// TIA Portal V19 export
FUNCTION "OUTPUT MAPPING" : Void   // FC2, LAD
{ S7_Optimized_Access := 'TRUE' }
// stored: SetENOAutomatically false
BEGIN

REGION Network 1: "HOOTER RESET"
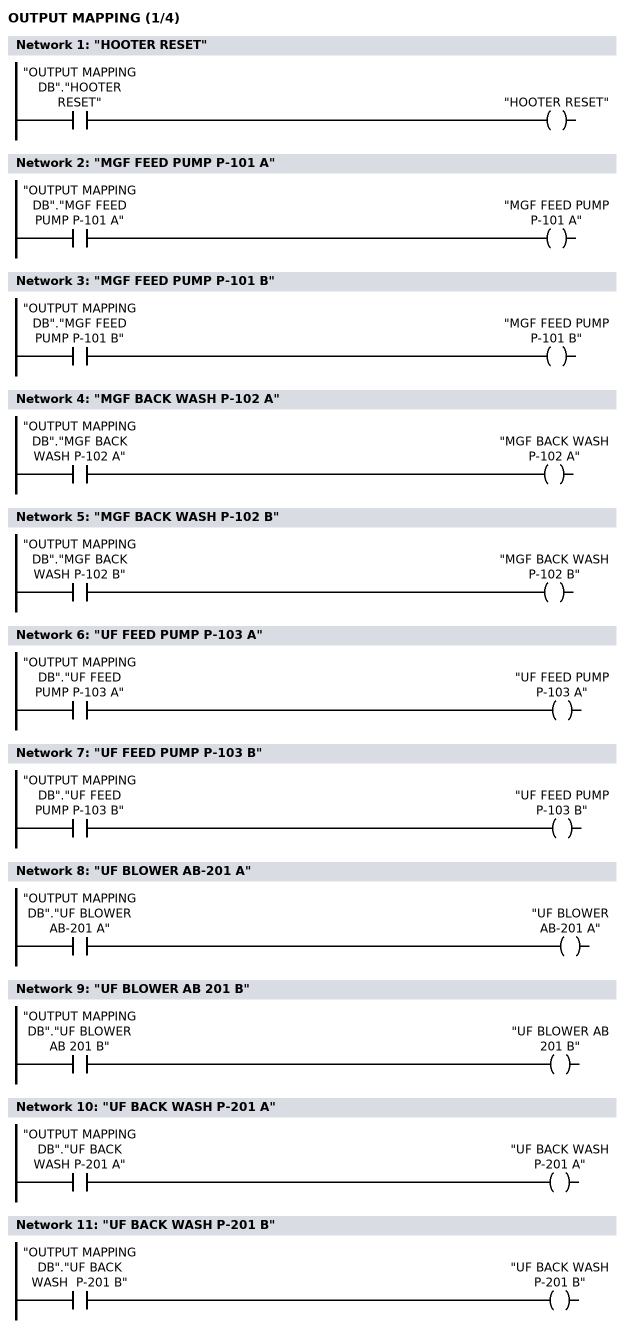
   RUNG wire#powerrail
      Contact( "OUTPUT MAPPING DB"."HOOTER RESET" )
      Coil( "HOOTER RESET" )
   END_RUNG
   // the same network as SCL:
   "HOOTER RESET" := "OUTPUT MAPPING DB"."HOOTER RESET";
END_REGION

REGION Network 2: "MGF FEED PUMP P-101 A"
   RUNG wire#powerrail
      Contact( "OUTPUT MAPPING DB"."MGF FEED PUMP P-101 A" )
      Coil( "MGF FEED PUMP P-101 A" )
   END_RUNG
   // the same network as SCL:
   "MGF FEED PUMP P-101 A" := "OUTPUT MAPPING DB"."MGF FEED PUMP P-101 A";
END_REGION

REGION Network 3: "MGF FEED PUMP P-101 B"
   RUNG wire#powerrail
      Contact( "OUTPUT MAPPING DB"."MGF FEED PUMP P-101 B" )
      Coil( "MGF FEED PUMP P-101 B" )
   END_RUNG
   // the same network as SCL:
   "MGF FEED PUMP P-101 B" := "OUTPUT MAPPING DB"."MGF FEED PUMP P-101 B";
END_REGION

REGION Network 4: "MGF BACK WASH P-102 A"
   RUNG wire#powerrail
      Contact( "OUTPUT MAPPING DB"."MGF BACK WASH P-102 A" )
      Coil( "MGF BACK WASH P-102 A" )
   END_RUNG
   // the same network as SCL:
   "MGF BACK WASH P-102 A" := "OUTPUT MAPPING DB"."MGF BACK WASH P-102 A";
END_REGION

REGION Network 5: "MGF BACK WASH P-102 B"
   RUNG wire#powerrail
      Contact( "OUTPUT MAPPING DB"."MGF BACK WASH P-102 B" )
      Coil( "MGF BACK WASH P-102 B" )
   END_RUNG
   // the same network as SCL:
   "MGF BACK WASH P-102 B" := "OUTPUT MAPPING DB"."MGF BACK WASH P-102 B";
END_REGION

REGION Network 6: "UF FEED PUMP P-103 A"
   RUNG wire#powerrail
      Contact( "OUTPUT MAPPING DB"."UF FEED PUMP P-103 A" )
      Coil( "UF FEED PUMP P-103 A" )
   END_RUNG
   // the same network as SCL:
   "UF FEED PUMP P-103 A" := "OUTPUT MAPPING DB"."UF FEED PUMP P-103 A";
END_REGION

REGION Network 7: "UF FEED PUMP P-103 B"
   RUNG wire#powerrail
      Contact( "OUTPUT MAPPING DB"."UF FEED PUMP P-103 B" )
      Coil( "UF FEED PUMP P-103 B" )
   END_RUNG
   // the same network as SCL:
   "UF FEED PUMP P-103 B" := "OUTPUT MAPPING DB"."UF FEED PUMP P-103 B";
END_REGION

REGION Network 8: "UF BLOWER AB-201 A"
   RUNG wire#powerrail
      Contact( "OUTPUT MAPPING DB"."UF BLOWER AB-201 A" )
      Coil( "UF BLOWER AB-201 A" )
   END_RUNG
   // the same network as SCL:
   "UF BLOWER AB-201 A" := "OUTPUT MAPPING DB"."UF BLOWER AB-201 A";
END_REGION

REGION Network 9: "UF BLOWER AB 201 B"
   RUNG wire#powerrail
      Contact( "OUTPUT MAPPING DB"."UF BLOWER AB 201 B" )
      Coil( "UF BLOWER AB 201 B" )
   END_RUNG
   // the same network as SCL:
   "UF BLOWER AB 201 B" := "OUTPUT MAPPING DB"."UF BLOWER AB 201 B";
END_REGION

REGION Network 10: "UF BACK WASH P-201 A"
   RUNG wire#powerrail
      Contact( "OUTPUT MAPPING DB"."UF BACK WASH P-201 A" )
      Coil( "UF BACK WASH P-201 A" )
   END_RUNG
   // the same network as SCL:
   "UF BACK WASH P-201 A" := "OUTPUT MAPPING DB"."UF BACK WASH P-201 A";
END_REGION

REGION Network 11: "UF BACK WASH P-201 B"
   RUNG wire#powerrail
      Contact( "OUTPUT MAPPING DB"."UF BACK WASH  P-201 B" )
      Coil( "UF BACK WASH  P-201 B" )
   END_RUNG
   // the same network as SCL:
   "UF BACK WASH  P-201 B" := "OUTPUT MAPPING DB"."UF BACK WASH  P-201 B";
END_REGION

REGION Network 12: "DM FEED PUMP P-502 A"
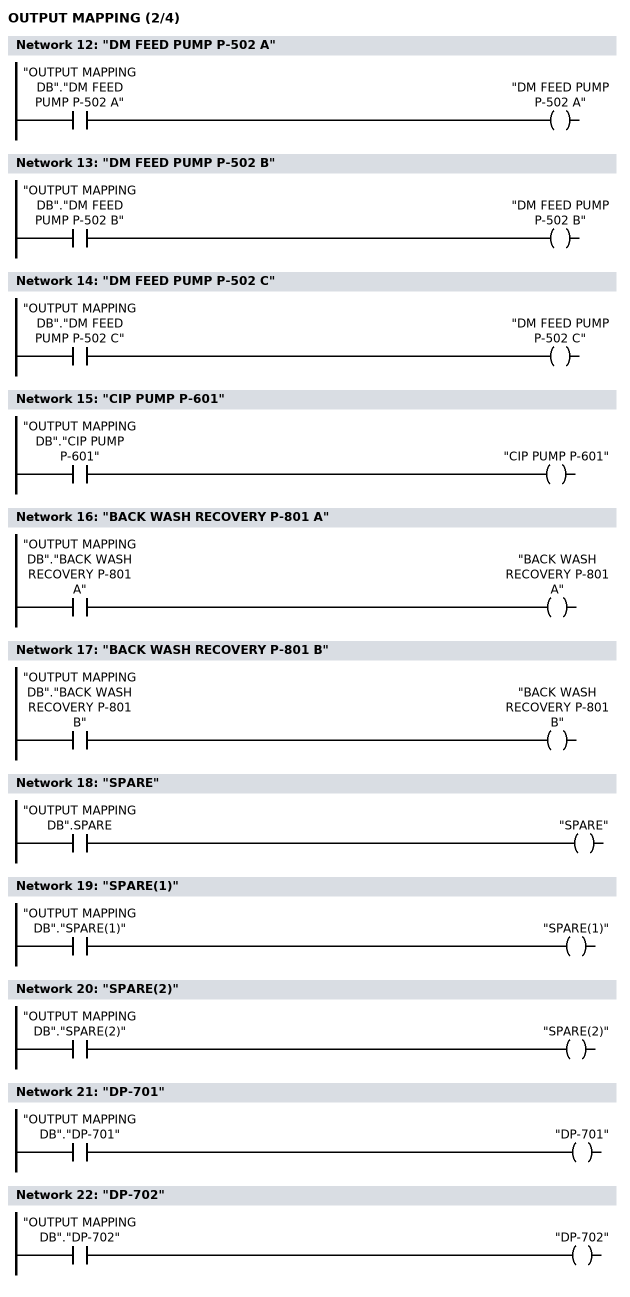
   RUNG wire#powerrail
      Contact( "OUTPUT MAPPING DB"."DM FEED PUMP P-502 A" )
      Coil( "DM FEED PUMP P-502 A" )
   END_RUNG
   // the same network as SCL:
   "DM FEED PUMP P-502 A" := "OUTPUT MAPPING DB"."DM FEED PUMP P-502 A";
END_REGION

REGION Network 13: "DM FEED PUMP P-502 B"
   RUNG wire#powerrail
      Contact( "OUTPUT MAPPING DB"."DM FEED PUMP P-502 B" )
      Coil( "DM FEED PUMP P-502 B" )
   END_RUNG
   // the same network as SCL:
   "DM FEED PUMP P-502 B" := "OUTPUT MAPPING DB"."DM FEED PUMP P-502 B";
END_REGION

REGION Network 14: "DM FEED PUMP P-502 C"
   RUNG wire#powerrail
      Contact( "OUTPUT MAPPING DB"."DM FEED PUMP P-502 C" )
      Coil( "DM FEED PUMP P-502 C" )
   END_RUNG
   // the same network as SCL:
   "DM FEED PUMP P-502 C" := "OUTPUT MAPPING DB"."DM FEED PUMP P-502 C";
END_REGION

REGION Network 15: "CIP PUMP P-601"
   RUNG wire#powerrail
      Contact( "OUTPUT MAPPING DB"."CIP PUMP P-601" )
      Coil( "CIP PUMP P-601" )
   END_RUNG
   // the same network as SCL:
   "CIP PUMP P-601" := "OUTPUT MAPPING DB"."CIP PUMP P-601";
END_REGION

REGION Network 16: "BACK WASH RECOVERY P-801 A"
   RUNG wire#powerrail
      Contact( "OUTPUT MAPPING DB"."BACK WASH RECOVERY P-801 A" )
      Coil( "BACK WASH RECOVERY P-801 A" )
   END_RUNG
   // the same network as SCL:
   "BACK WASH RECOVERY P-801 A" := "OUTPUT MAPPING DB"."BACK WASH RECOVERY P-801 A";
END_REGION

REGION Network 17: "BACK WASH RECOVERY P-801 B"
   RUNG wire#powerrail
      Contact( "OUTPUT MAPPING DB"."BACK WASH RECOVERY P-801 B" )
      Coil( "BACK WASH RECOVERY P-801 B" )
   END_RUNG
   // the same network as SCL:
   "BACK WASH RECOVERY P-801 B" := "OUTPUT MAPPING DB"."BACK WASH RECOVERY P-801 B";
END_REGION

REGION Network 18: "SPARE"
   RUNG wire#powerrail
      Contact( "OUTPUT MAPPING DB".SPARE )
      Coil( "SPARE" )
   END_RUNG
   // the same network as SCL:
   "SPARE" := "OUTPUT MAPPING DB".SPARE;
END_REGION

REGION Network 19: "SPARE(1)"
   RUNG wire#powerrail
      Contact( "OUTPUT MAPPING DB"."SPARE(1)" )
      Coil( "SPARE(1)" )
   END_RUNG
   // the same network as SCL:
   "SPARE(1)" := "OUTPUT MAPPING DB"."SPARE(1)";
END_REGION

REGION Network 20: "SPARE(2)"
   RUNG wire#powerrail
      Contact( "OUTPUT MAPPING DB"."SPARE(2)" )
      Coil( "SPARE(2)" )
   END_RUNG
   // the same network as SCL:
   "SPARE(2)" := "OUTPUT MAPPING DB"."SPARE(2)";
END_REGION

REGION Network 21: "DP-701"
   RUNG wire#powerrail
      Contact( "OUTPUT MAPPING DB"."DP-701" )
      Coil( "DP-701" )
   END_RUNG
   // the same network as SCL:
   "DP-701" := "OUTPUT MAPPING DB"."DP-701";
END_REGION

REGION Network 22: "DP-702"
   RUNG wire#powerrail
      Contact( "OUTPUT MAPPING DB"."DP-702" )
      Coil( "DP-702" )
   END_RUNG
   // the same network as SCL:
   "DP-702" := "OUTPUT MAPPING DB"."DP-702";
END_REGION

REGION Network 23: "NaOCL DOSING D-706 A"
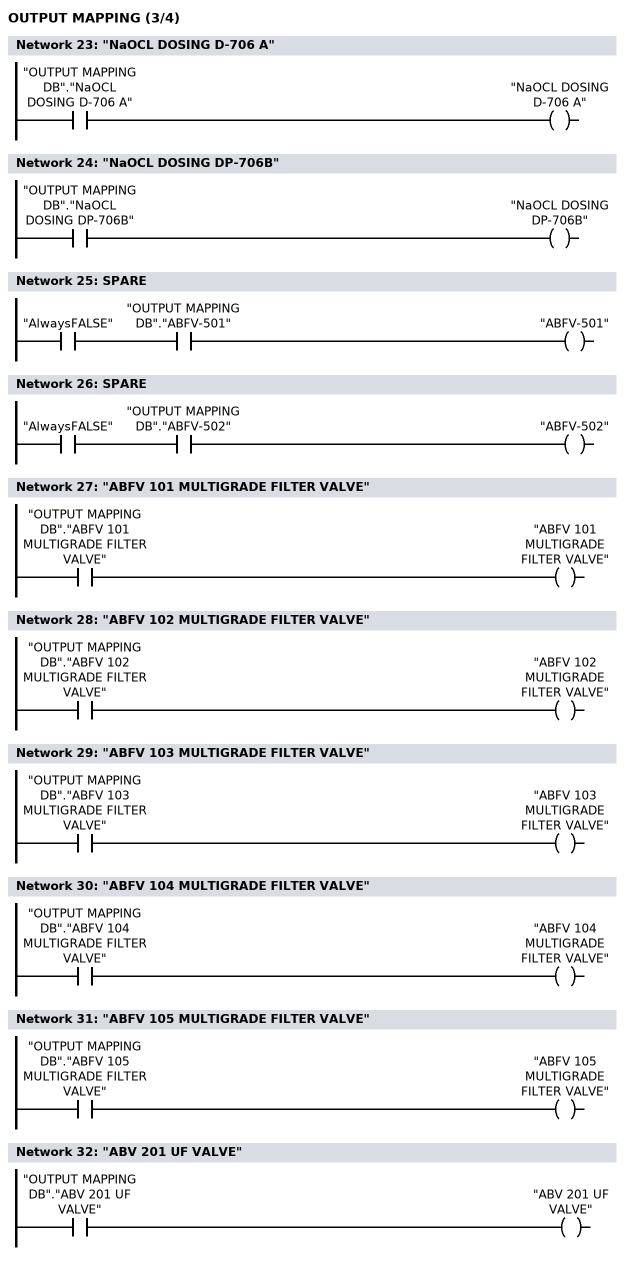
   RUNG wire#powerrail
      Contact( "OUTPUT MAPPING DB"."NaOCL DOSING D-706 A" )
      Coil( "NaOCL DOSING D-706 A" )
   END_RUNG
   // the same network as SCL:
   "NaOCL DOSING D-706 A" := "OUTPUT MAPPING DB"."NaOCL DOSING D-706 A";
END_REGION

REGION Network 24: "NaOCL DOSING DP-706B"
   RUNG wire#powerrail
      Contact( "OUTPUT MAPPING DB"."NaOCL DOSING DP-706B" )
      Coil( "NaOCL DOSING DP-706B" )
   END_RUNG
   // the same network as SCL:
   "NaOCL DOSING DP-706B" := "OUTPUT MAPPING DB"."NaOCL DOSING DP-706B";
END_REGION

REGION Network 25: SPARE
   RUNG wire#powerrail
      Contact( "AlwaysFALSE" )
      Contact( "OUTPUT MAPPING DB"."ABFV-501" )
      Coil( "ABFV-501" )
   END_RUNG
   // the same network as SCL:
   "ABFV-501" := "AlwaysFALSE" AND "OUTPUT MAPPING DB"."ABFV-501";
END_REGION

REGION Network 26: SPARE
   RUNG wire#powerrail
      Contact( "AlwaysFALSE" )
      Contact( "OUTPUT MAPPING DB"."ABFV-502" )
      Coil( "ABFV-502" )
   END_RUNG
   // the same network as SCL:
   "ABFV-502" := "AlwaysFALSE" AND "OUTPUT MAPPING DB"."ABFV-502";
END_REGION

REGION Network 27: "ABFV 101 MULTIGRADE FILTER VALVE"
   RUNG wire#powerrail
      Contact( "OUTPUT MAPPING DB"."ABFV 101 MULTIGRADE FILTER VALVE" )
      Coil( "ABFV 101 MULTIGRADE FILTER VALVE" )
   END_RUNG
   // the same network as SCL:
   "ABFV 101 MULTIGRADE FILTER VALVE" := "OUTPUT MAPPING DB"."ABFV 101 MULTIGRADE FILTER VALVE";
END_REGION

REGION Network 28: "ABFV 102 MULTIGRADE FILTER VALVE"
   RUNG wire#powerrail
      Contact( "OUTPUT MAPPING DB"."ABFV 102 MULTIGRADE FILTER VALVE" )
      Coil( "ABFV 102 MULTIGRADE FILTER VALVE" )
   END_RUNG
   // the same network as SCL:
   "ABFV 102 MULTIGRADE FILTER VALVE" := "OUTPUT MAPPING DB"."ABFV 102 MULTIGRADE FILTER VALVE";
END_REGION

REGION Network 29: "ABFV 103 MULTIGRADE FILTER VALVE"
   RUNG wire#powerrail
      Contact( "OUTPUT MAPPING DB"."ABFV 103 MULTIGRADE FILTER VALVE" )
      Coil( "ABFV 103 MULTIGRADE FILTER VALVE" )
   END_RUNG
   // the same network as SCL:
   "ABFV 103 MULTIGRADE FILTER VALVE" := "OUTPUT MAPPING DB"."ABFV 103 MULTIGRADE FILTER VALVE";
END_REGION

REGION Network 30: "ABFV 104 MULTIGRADE FILTER VALVE"
   RUNG wire#powerrail
      Contact( "OUTPUT MAPPING DB"."ABFV 104 MULTIGRADE FILTER VALVE" )
      Coil( "ABFV 104 MULTIGRADE FILTER VALVE" )
   END_RUNG
   // the same network as SCL:
   "ABFV 104 MULTIGRADE FILTER VALVE" := "OUTPUT MAPPING DB"."ABFV 104 MULTIGRADE FILTER VALVE";
END_REGION

REGION Network 31: "ABFV 105 MULTIGRADE FILTER VALVE"
   RUNG wire#powerrail
      Contact( "OUTPUT MAPPING DB"."ABFV 105 MULTIGRADE FILTER VALVE" )
      Coil( "ABFV 105 MULTIGRADE FILTER VALVE" )
   END_RUNG
   // the same network as SCL:
   "ABFV 105 MULTIGRADE FILTER VALVE" := "OUTPUT MAPPING DB"."ABFV 105 MULTIGRADE FILTER VALVE";
END_REGION

REGION Network 32: "ABV 201 UF VALVE"
   RUNG wire#powerrail
      Contact( "OUTPUT MAPPING DB"."ABV 201 UF VALVE" )
      Coil( "ABV 201 UF VALVE" )
   END_RUNG
   // the same network as SCL:
   "ABV 201 UF VALVE" := "OUTPUT MAPPING DB"."ABV 201 UF VALVE";
END_REGION

REGION Network 33: "ABFV 201 UF VALVE"
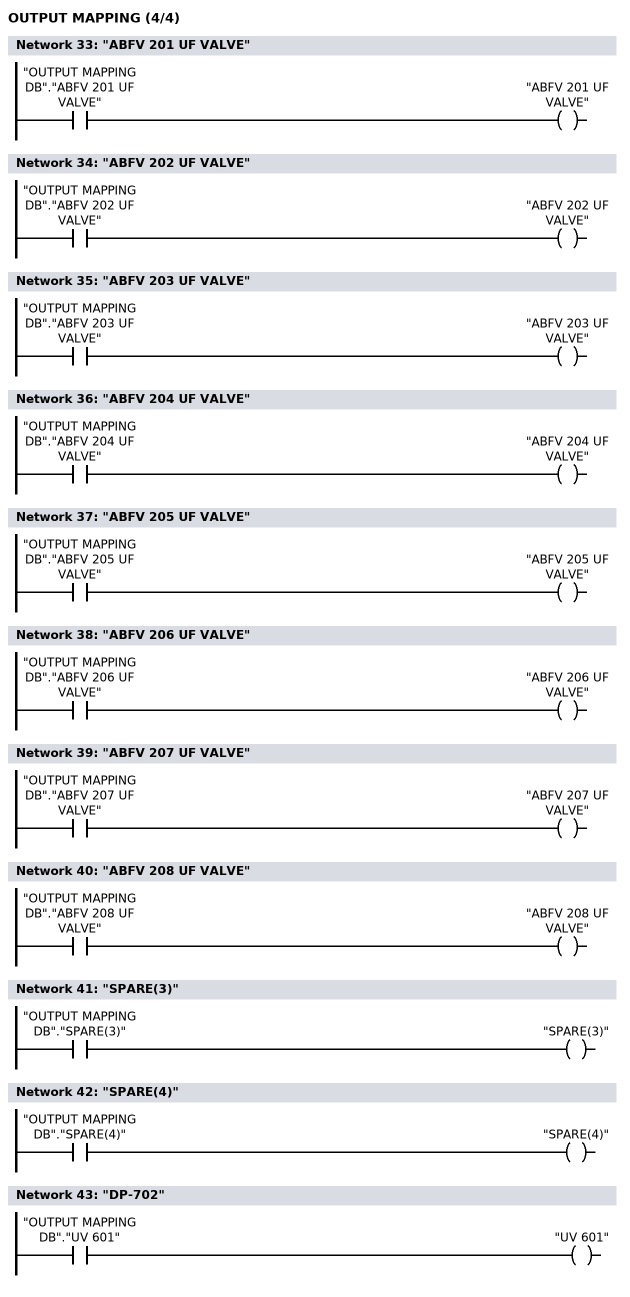
   RUNG wire#powerrail
      Contact( "OUTPUT MAPPING DB"."ABFV 201 UF VALVE" )
      Coil( "ABFV 201 UF VALVE" )
   END_RUNG
   // the same network as SCL:
   "ABFV 201 UF VALVE" := "OUTPUT MAPPING DB"."ABFV 201 UF VALVE";
END_REGION

REGION Network 34: "ABFV 202 UF VALVE"
   RUNG wire#powerrail
      Contact( "OUTPUT MAPPING DB"."ABFV 202 UF VALVE" )
      Coil( "ABFV 202 UF VALVE" )
   END_RUNG
   // the same network as SCL:
   "ABFV 202 UF VALVE" := "OUTPUT MAPPING DB"."ABFV 202 UF VALVE";
END_REGION

REGION Network 35: "ABFV 203 UF VALVE"
   RUNG wire#powerrail
      Contact( "OUTPUT MAPPING DB"."ABFV 203 UF VALVE" )
      Coil( "ABFV 203 UF VALVE" )
   END_RUNG
   // the same network as SCL:
   "ABFV 203 UF VALVE" := "OUTPUT MAPPING DB"."ABFV 203 UF VALVE";
END_REGION

REGION Network 36: "ABFV 204 UF VALVE"
   RUNG wire#powerrail
      Contact( "OUTPUT MAPPING DB"."ABFV 204 UF VALVE" )
      Coil( "ABFV 204 UF VALVE" )
   END_RUNG
   // the same network as SCL:
   "ABFV 204 UF VALVE" := "OUTPUT MAPPING DB"."ABFV 204 UF VALVE";
END_REGION

REGION Network 37: "ABFV 205 UF VALVE"
   RUNG wire#powerrail
      Contact( "OUTPUT MAPPING DB"."ABFV 205 UF VALVE" )
      Coil( "ABFV 205 UF VALVE" )
   END_RUNG
   // the same network as SCL:
   "ABFV 205 UF VALVE" := "OUTPUT MAPPING DB"."ABFV 205 UF VALVE";
END_REGION

REGION Network 38: "ABFV 206 UF VALVE"
   RUNG wire#powerrail
      Contact( "OUTPUT MAPPING DB"."ABFV 206 UF VALVE" )
      Coil( "ABFV 206 UF VALVE" )
   END_RUNG
   // the same network as SCL:
   "ABFV 206 UF VALVE" := "OUTPUT MAPPING DB"."ABFV 206 UF VALVE";
END_REGION

REGION Network 39: "ABFV 207 UF VALVE"
   RUNG wire#powerrail
      Contact( "OUTPUT MAPPING DB"."ABFV 207 UF VALVE" )
      Coil( "ABFV 207 UF VALVE" )
   END_RUNG
   // the same network as SCL:
   "ABFV 207 UF VALVE" := "OUTPUT MAPPING DB"."ABFV 207 UF VALVE";
END_REGION

REGION Network 40: "ABFV 208 UF VALVE"
   RUNG wire#powerrail
      Contact( "OUTPUT MAPPING DB"."ABFV 208 UF VALVE" )
      Coil( "ABFV 208 UF VALVE" )
   END_RUNG
   // the same network as SCL:
   "ABFV 208 UF VALVE" := "OUTPUT MAPPING DB"."ABFV 208 UF VALVE";
END_REGION

REGION Network 41: "SPARE(3)"
   RUNG wire#powerrail
      Contact( "OUTPUT MAPPING DB"."SPARE(3)" )
      Coil( "SPARE(3)" )
   END_RUNG
   // the same network as SCL:
   "SPARE(3)" := "OUTPUT MAPPING DB"."SPARE(3)";
END_REGION

REGION Network 42: "SPARE(4)"
   RUNG wire#powerrail
      Contact( "OUTPUT MAPPING DB"."SPARE(4)" )
      Coil( "SPARE(4)" )
   END_RUNG
   // the same network as SCL:
   "SPARE(4)" := "OUTPUT MAPPING DB"."SPARE(4)";
END_REGION

REGION Network 43: "DP-702"
   RUNG wire#powerrail
      Contact( "OUTPUT MAPPING DB"."UV 601" )
      Coil( "UV 601" )
   END_RUNG
   // the same network as SCL:
   "UV 601" := "OUTPUT MAPPING DB"."UV 601";
END_REGION
END_FUNCTION
